FUNCTION_BLOCK MoveMoverToPosition EXTENDS TaskBase
VAR_INPUT
END_VAR
VAR_OUTPUT
END_VAR
VAR
	moveAbs	: MC_MoveAbsoluteCA;
	_Axis : REFERENCE TO AXIS_REF;
	_MoveMover : BOOL;
	_stOptions : ST_MoveAbsoluteCAOptions;
END_VAR

{analysis -2}

METHOD Abort : BOOL
moveAbs.Execute := FALSE;
moveAbs.Position := moveAbs.Velocity := 0;
_MoveMover := false;
_Busy := FALSE;
Abort := true;
State := 0;
END_METHOD

PROPERTY PUBLIC Acceleration : mc_lreal
GET
Acceleration := moveAbs.Acceleration;
END_GET
SET
moveAbs.Acceleration := Acceleration;
END_SET
END_PROPERTY

METHOD Cycle : HRESULT
VAR_INPUT
END_VAR
CASE State OF
	0:
		IF _MoveMover THEN
			Cycle := S_PENDING;
			_Done := FALSE;
			_Error := FALSE;
			_Busy := TRUE;
			moveAbs.Execute := TRUE;
			IF moveAbs.Busy THEN
				State := 10;
				_MoveMover := FALSE;
			END_IF
		END_IF
		
	10:
		IF NOT moveAbs.Busy THEN
			IF moveAbs.Done THEN
				_Done := TRUE;
			ELSIF moveAbs.Error THEN
				_Error := TRUE;
			END_IF
			_Busy := FALSE;
			moveAbs.Execute := FALSE;
			State := 0;
			Cycle := S_OK;
		END_IF
END_CASE

moveAbs(Axis := _Axis, Options := _stOptions);
END_METHOD

PROPERTY PUBLIC Deceleration : mc_lreal
GET
Deceleration := moveAbs.Deceleration;
END_GET
SET
moveAbs.Deceleration := Deceleration;
END_SET
END_PROPERTY

METHOD FB_init : BOOL
VAR_INPUT
	bInitRetains : BOOL; // if TRUE, the retain variables are initialized (warm start / cold start)
	bInCopyCode : BOOL;  // if TRUE, the instance afterwards gets moved into the copy code (online change)
	axis : reference TO AXIS_REF;
END_VAR
_Axis REF= axis;
END_METHOD

PROPERTY PUBLIC Gap : mc_lreal
GET
Gap := moveAbs.Gap;
END_GET
SET
moveAbs.Gap := Gap;
END_SET
END_PROPERTY

PROPERTY PUBLIC Jerk : mc_lreal
GET
Jerk := moveAbs.Jerk;
END_GET
SET
moveAbs.Jerk := Jerk;
END_SET
END_PROPERTY

METHOD MoveTo : BOOL
VAR_INPUT
	Position : MC_LREAL;
	Velocity : MC_LREAL;
END_VAR
moveAbs.Position := Position;
moveAbs.Velocity := Velocity;
_MoveMover := MoveTo := true;
END_METHOD

PROPERTY PUBLIC Options : ST_MoveAbsoluteCAOptions
GET
Options := _stOptions;
END_GET
SET
_stOptions := Options;
END_SET
END_PROPERTY

END_FUNCTION_BLOCK

(* stored: Version 1.1.0.1, ProductVersion 3.1.4024.12
   POU MoveMoverToPosition: Id {3c31ca33-c741-4f8c-92b8-6b6baade4c31}, SpecialFunc None
   Method Abort: Id {7dbf4838-5de6-4b26-9062-b550522ba980}
   Property Acceleration: Id {1b0568fa-dc0f-4b6a-9678-65b35bd8e086}
   Get Get: Id {3269a981-3cbd-416a-9174-686fb77d432b}
   Set Set: Id {26ebe242-b19a-49f2-b37a-99cd788cb644}
   Method Cycle: Id {237a9ac8-3d0d-42a7-bef7-613d3b5a1246}
   Property Deceleration: Id {712ea7f9-753f-4107-9079-a1664cc0d22a}
   Get Get: Id {ae3fd434-8e55-45d4-8b26-cf54b665b9fb}
   Set Set: Id {61ceb198-6fa9-42b7-8ec0-d722e08d8888}
   Method FB_init: Id {83f57c14-6be4-4377-9659-d2815ee74447}
   Property Gap: Id {963f9ec5-5fa3-4be4-84c6-11ed60e6d70b}
   Get Get: Id {4720dd6a-d593-4539-aa5e-5f86357c18d6}
   Set Set: Id {6a524761-7858-4e5b-86be-235454598954}
   Property Jerk: Id {824794e9-2a38-44d5-b5b0-9429ee22fdef}
   Get Get: Id {9fc03e76-309c-42bf-a7cb-98a28ba166ac}
   Set Set: Id {ea7b06e9-acb9-44db-a7b6-cf0cb4c35d8c}
   Method MoveTo: Id {7a988821-6187-410c-9f44-ac37dd79e4ea}
   Property Options: Id {dea942d2-1849-46bc-9a6f-e7e95c9dca3d}
   Get Get: Id {a992cdcd-3d01-465b-8643-1084be02841d}
   Set Set: Id {0dae0639-08f2-4a8c-85bd-6d17b1e1285f} *)
